KUKA KRL program: CHEQUEO_GARRA.src, CHEQUEO_GARRA.dat

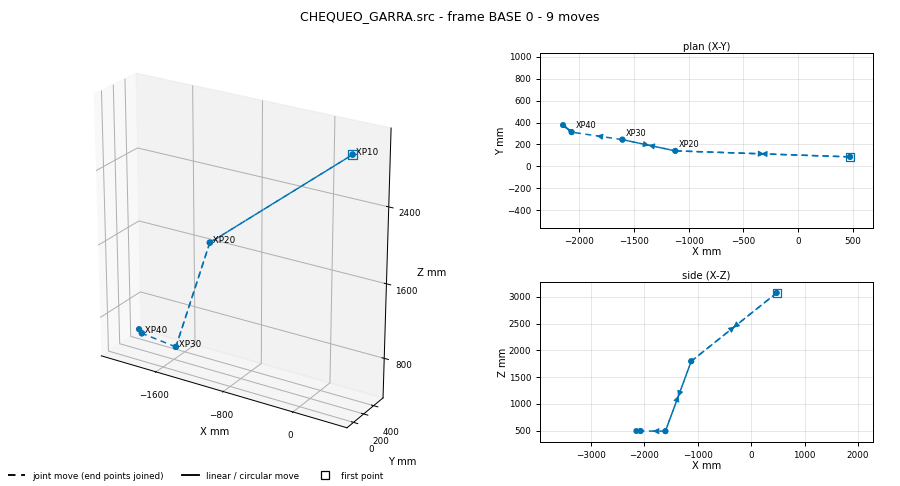
[picture p0: tool path of CHEQUEO_GARRA.src in frame BASE 0, 9 of 12 moves have a stored position in this frame; points joined in program order, loops and branches not executed]
--- CHEQUEO_GARRA.src ---
&ACCESS RVO1
&REL 10
&COMMENT PRG CONTROL GARRA
&PARAM EDITMASK = *
&PARAM TEMPLATE = C:\KRC\Roboter\Template\vorgabe
&PARAM DISKPATH = KRC:\R1\Program\MAFELEC
DEF CHEQUEO_GARRA( )
;FOLD INI;%{PE}
  ;FOLD BASISTECH INI
    GLOBAL INTERRUPT DECL 3 WHEN $STOPMESS==TRUE DO IR_STOPM ( )
    INTERRUPT ON 3
    BAS (#INITMOV,0 )
  ;ENDFOLD (BASISTECH INI)
;FOLD SPOTTECH INI
USERSPOT(#INIT)
;ENDFOLD (SPOTTECH INI)
;FOLD GRIPPERTECH INI
USER_GRP(0,DUMMY,DUMMY,GDEFAULT)
;ENDFOLD (GRIPPERTECH INI)
  ;FOLD USER INI
    ;Make your modifications here

  ;ENDFOLD (USER INI)
;ENDFOLD (INI)
;################################################
; PROYECTO: MAFELEC PLANTA DE BATERIAS
; ROBOT: 121_R1
; PROGRAMA: CHEQUEO EN GALGA DE CONTROL GARRA
; CREADO POR: La Rosaliaaaa(zaisor robotics)
; FECHA: 28-NOVIEMBRE-2022
; MODIFICADO POR:
; FECHA MODIFICACION: 9-ENERO-2023
;################################################

;FOLD PTP HOME  Vel= 100 % DEFAULT;%{PE}%MKUKATPBASIS,%CMOVE,%VPTP,%P 1:PTP, 2:HOME, 3:, 5:100, 7:DEFAULT
$BWDSTART = FALSE
PDAT_ACT=PDEFAULT
FDAT_ACT=FHOME
BAS (#PTP_PARAMS,100 )
$H_POS=XHOME
PTP  XHOME
;ENDFOLD

Empujador(1,"R",TRUE)
Empujador(2,"R",TRUE)
Pines("R")

;FOLD PTP P10 CONT Vel=100 % M Tool[9]:T_Gripper1_Vacio Base[0];%{PE}%R 8.3.48,%MKUKATPBASIS,%CMOVE,%VPTP,%P 1:PTP, 2:P10, 3:C_DIS, 5:100, 7:M
$BWDSTART=FALSE
PDAT_ACT=PM
FDAT_ACT=FP10
BAS(#PTP_PARAMS,100)
PTP XP10 C_DIS
;ENDFOLD
;FOLD PTP P20 CONT Vel=100 % M Tool[9]:T_Gripper1_Vacio Base[0];%{PE}%R 8.3.48,%MKUKATPBASIS,%CMOVE,%VPTP,%P 1:PTP, 2:P20, 3:C_DIS, 5:100, 7:M
$BWDSTART=FALSE
PDAT_ACT=PM
FDAT_ACT=FP20
BAS(#PTP_PARAMS,100)
PTP XP20 C_DIS
;ENDFOLD
;FOLD PTP P30 CONT Vel=100 % M Tool[9]:T_Gripper1_Vacio Base[0];%{PE}%R 8.3.48,%MKUKATPBASIS,%CMOVE,%VPTP,%P 1:PTP, 2:P30, 3:C_DIS, 5:100, 7:M
$BWDSTART=FALSE
PDAT_ACT=PM
FDAT_ACT=FP30
BAS(#PTP_PARAMS,100)
PTP XP30 C_DIS
;ENDFOLD
;FOLD PTP P40 CONT Vel=100 % M Tool[9]:T_Gripper1_Vacio Base[0];%{PE}%R 8.3.48,%MKUKATPBASIS,%CMOVE,%VPTP,%P 1:PTP, 2:P40, 3:C_DIS, 5:100, 7:M
$BWDSTART=FALSE
PDAT_ACT=PM
FDAT_ACT=FP40
BAS(#PTP_PARAMS,100)
PTP XP40 C_DIS
;ENDFOLD

; FOLD ESPERA LLAVE EN MANUAL(T1),CONTROLAR GARRA EN GALGA
Pines("R")
WAIT FOR $T1
;ENDFOLD

;FOLD LIN POSICION_CONTROL Vel=0.1 m/s M Tool[9]:T_Gripper1_Vacio Base[0];%{PE}%R 8.3.48,%MKUKATPBASIS,%CMOVE,%VLIN,%P 1:LIN, 2:POSICION_CONTROL, 3:, 5:0.1, 7:M
$BWDSTART=FALSE
LDAT_ACT=LM
FDAT_ACT=FPOSICION_CONTROL
BAS(#CP_PARAMS,0.1)
LIN XPOSICION_CONTROL
;ENDFOLD

;Pines("A")
O_121R1Y13B=FALSE
O_121R1Y13A=TRUE
O_121R1Y132B=FALSE
O_121R1Y132A=TRUE

WAIT FOR (I_121R1S131A AND I_121R1S132A AND I_121R1S133A AND I_121R1S134A)
WAIT SEC 10
Pines("R")


;FOLD LIN P40 Vel=0.5 m/s M Tool[9]:T_Gripper1_Vacio Base[0];%{PE}%R 8.3.48,%MKUKATPBASIS,%CMOVE,%VLIN,%P 1:LIN, 2:P40, 3:, 5:0.5, 7:M
$BWDSTART=FALSE
LDAT_ACT=LM
FDAT_ACT=FP40
BAS(#CP_PARAMS,0.5)
LIN XP40
;ENDFOLD

;FOLD CAMBIAR LA LLAVE A EXT Y CONTINUAR
Pines("R")
PTP $POS_ACT
WAIT FOR $EXT
Pines("R")
;ENDFOLD

;FOLD PTP P30 CONT Vel=100 % M Tool[9]:T_Gripper1_Vacio Base[0];%{PE}%R 8.3.48,%MKUKATPBASIS,%CMOVE,%VPTP,%P 1:PTP, 2:P30, 3:C_DIS, 5:100, 7:M
$BWDSTART=FALSE
PDAT_ACT=PM
FDAT_ACT=FP30
BAS(#PTP_PARAMS,100)
PTP XP30 C_DIS
;ENDFOLD
;FOLD PTP P20 CONT Vel=100 % M Tool[9]:T_Gripper1_Vacio Base[0];%{PE}%R 8.3.48,%MKUKATPBASIS,%CMOVE,%VPTP,%P 1:PTP, 2:P20, 3:C_DIS, 5:100, 7:M
$BWDSTART=FALSE
PDAT_ACT=PM
FDAT_ACT=FP20
BAS(#PTP_PARAMS,100)
PTP XP20 C_DIS
;ENDFOLD
;FOLD PTP P10 CONT Vel=100 % M Tool[9]:T_Gripper1_Vacio Base[0];%{PE}%R 8.3.48,%MKUKATPBASIS,%CMOVE,%VPTP,%P 1:PTP, 2:P10, 3:C_DIS, 5:100, 7:M
$BWDSTART=FALSE
PDAT_ACT=PM
FDAT_ACT=FP10
BAS(#PTP_PARAMS,100)
PTP XP10 C_DIS
;ENDFOLD

;FOLD PTP HOME  Vel= 100 % DEFAULT;%{PE}%MKUKATPBASIS,%CMOVE,%VPTP,%P 1:PTP, 2:HOME, 3:, 5:100, 7:DEFAULT
$BWDSTART = FALSE
PDAT_ACT=PDEFAULT
FDAT_ACT=FHOME
BAS (#PTP_PARAMS,100 )
$H_POS=XHOME
PTP  XHOME
;ENDFOLD

END

--- CHEQUEO_GARRA.dat ---
&ACCESS RVO1
&REL 10
&COMMENT PRG CONTROL GARRA
&PARAM EDITMASK = *
&PARAM TEMPLATE = C:\KRC\Roboter\Template\vorgabe
&PARAM DISKPATH = KRC:\R1\Program\MAFELEC
DEFDAT  CHEQUEO_GARRA
;FOLD EXTERNAL DECLARATIONS;%{PE}%MKUKATPBASIS,%CEXT,%VCOMMON,%P
;FOLD GRIPPERTECH EXT
EXT  H50 (INT  :IN,INT  :IN,INT  :IN,GRP_TYP  :IN )
;ENDFOLD (GRIPPERTECH EXT)
;FOLD SPOTTECH EXT
EXT  USERSPOT (S_COMMAND  :IN,SPOT_TYPE  :IN )
;ENDFOLD (SPOTTECH EXT)
;FOLD BASISTECH EXT;%{PE}%MKUKATPBASIS,%CEXT,%VEXT,%P
EXT  BAS (BAS_COMMAND  :IN,REAL  :IN )
DECL INT SUCCESS
;ENDFOLD (BASISTECH EXT)
;FOLD USER EXT;%{E}%MKUKATPUSER,%CEXT,%VEXT,%P
;Make your modifications here

;ENDFOLD (USER EXT)
;ENDFOLD (EXTERNAL DECLARATIONS)
DECL BASIS_SUGG_T LAST_BASIS={POINT1[] "P43                     ",POINT2[] "P43                     ",CP_PARAMS[] "M                       ",PTP_PARAMS[] "M                       ",CONT[] "                        ",CP_VEL[] "0.1                     ",PTP_VEL[] "100                     ",SYNC_PARAMS[] "SYNCDAT                 ",SPL_NAME[] "S0                      ",A_PARAMS[] "ADAT0                   "}
DECL E6POS XP1={X -1423.22278,Y 12.1733541,Z 595.070862,A 13.3003607,B 1.31921577,C -179.688721,S 2,T 11,E1 0.0,E2 0.0,E3 0.0,E4 0.0,E5 0.0,E6 0.0}
DECL FDAT FP1={TOOL_NO 9,BASE_NO 0,IPO_FRAME #BASE,POINT2[] " ",TQ_STATE FALSE}
DECL PDAT PPDAT1={VEL 100.000,ACC 100.000,APO_DIST 100.000,APO_MODE #CDIS,GEAR_JERK 50.0000,EXAX_IGN 0}
DECL E6POS XP10={X 477.041595,Y 86.2656479,Z 3074.07861,A -151.431854,B -26.5239220,C 5.04246378,S 7,T 27,E1 0.0,E2 0.0,E3 0.0,E4 0.0,E5 0.0,E6 0.0}
DECL FDAT FP10={TOOL_NO 9,BASE_NO 0,IPO_FRAME #BASE,POINT2[] " ",TQ_STATE FALSE}
DECL E6POS XP20={X -1121.23938,Y 141.131592,Z 1796.16418,A 82.8106613,B 27.3655396,C -60.9739914,S 6,T 27,E1 0.0,E2 0.0,E3 0.0,E4 0.0,E5 0.0,E6 0.0}
DECL FDAT FP20={TOOL_NO 9,BASE_NO 0,IPO_FRAME #BASE,POINT2[] " ",TQ_STATE FALSE}
DECL PDAT PM={VEL 100.000,ACC 50.0000,APO_DIST 100.000,APO_MODE #CDIS,GEAR_JERK 50.0000,EXAX_IGN 0}
DECL E6POS XP30={X -1604.65100,Y 243.872147,Z 487.199,A 54.3264389,B -0.0970880091,C -89.6107407,S 6,T 27,E1 0.0,E2 0.0,E3 0.0,E4 0.0,E5 0.0,E6 0.0}
DECL FDAT FP30={TOOL_NO 9,BASE_NO 0,IPO_FRAME #BASE,POINT2[] " ",TQ_STATE FALSE}
DECL E6POS XP40={X -2068.92114,Y 312.188293,Z 491.154541,A 54.3907814,B 0.266583413,C -89.7929611,S 6,T 27,E1 0.0,E2 0.0,E3 0.0,E4 0.0,E5 0.0,E6 0.0}
DECL FDAT FP40={TOOL_NO 9,BASE_NO 0,IPO_FRAME #BASE,POINT2[] " ",TQ_STATE FALSE}
DECL E6POS XPOSICION_CONTROL={X -2148.42798,Y 377.520447,Z 490.690552,A 54.3906174,B 0.267401129,C -89.7934418,S 6,T 27,E1 0.0,E2 0.0,E3 0.0,E4 0.0,E5 0.0,E6 0.0}
DECL FDAT FPOSICION_CONTROL={TOOL_NO 9,BASE_NO 0,IPO_FRAME #BASE,POINT2[] " ",TQ_STATE FALSE}
DECL LDAT LM={VEL 2.00000,ACC 25.0000,APO_DIST 100.000,APO_FAC 50.0000,AXIS_VEL 100.000,AXIS_ACC 100.000,ORI_TYP #VAR,CIRC_TYP #BASE,JERK_FAC 50.0000,GEAR_JERK 50.0000,EXAX_IGN 0}
DECL E6POS XP41={X -1423.22278,Y 12.1733541,Z 595.070862,A 13.3003607,B 1.31921577,C -179.688721,S 2,T 11,E1 0.0,E2 0.0,E3 0.0,E4 0.0,E5 0.0,E6 0.0}
DECL FDAT FP41={TOOL_NO 9,BASE_NO 0,IPO_FRAME #BASE,POINT2[] " ",TQ_STATE FALSE}
DECL E6POS XP42={X -1423.22278,Y 12.1733541,Z 595.070862,A 13.3003607,B 1.31921577,C -179.688721,S 2,T 11,E1 0.0,E2 0.0,E3 0.0,E4 0.0,E5 0.0,E6 0.0}
DECL FDAT FP42={TOOL_NO 9,BASE_NO 0,IPO_FRAME #BASE,POINT2[] " ",TQ_STATE FALSE}
DECL E6POS XP43={X -1423.22278,Y 12.1733541,Z 595.070862,A 13.3003607,B 1.31921577,C -179.688721,S 2,T 11,E1 0.0,E2 0.0,E3 0.0,E4 0.0,E5 0.0,E6 0.0}
DECL FDAT FP43={TOOL_NO 9,BASE_NO 0,IPO_FRAME #BASE,POINT2[] " ",TQ_STATE FALSE}
ENDDAT
